FUNCTION_BLOCK FlushGritScreenCond (* Basic Function Block Type *)
  (* Standard: 61499-2 *)
  (* Version 0.0, 5/26/2024, SESA713705, Schneider Electric, Template *)
  PACKAGE SE.Nereda;
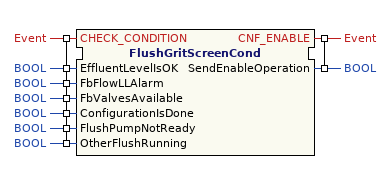
  EVENT_INPUT
    CHECK_CONDITION WITH EffluentLevelIsOK, FbFlowLLAlarm, FbValvesAvailable, ConfigurationIsDone, FlushPumpNotReady, OtherFlushRunning;
  END_EVENT
  EVENT_OUTPUT
    CNF_ENABLE WITH SendEnableOperation; (* Execution Confirmation *)
  END_EVENT
  VAR_INPUT
    EffluentLevelIsOK : BOOL;
    FbFlowLLAlarm : BOOL;
    FbValvesAvailable : BOOL;
    ConfigurationIsDone : BOOL;
    FlushPumpNotReady : BOOL;
    OtherFlushRunning : BOOL;
  END_VAR
  VAR_OUTPUT
    SendEnableOperation : BOOL;
  END_VAR
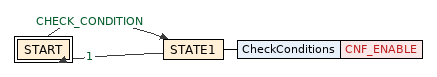
  EC_STATES
    START; (* Initial State *)
    STATE1 : CheckConditions -> CNF_ENABLE;
  END_STATES
  EC_TRANSITIONS
    START TO STATE1 := CHECK_CONDITION;
    STATE1 TO START := 1;
  END_TRANSITIONS
  ALGORITHM CheckConditions IN ST:
;
IF 	EffluentLevelIsOK = TRUE AND
	FbFlowLLAlarm = FALSE AND
	FbValvesAvailable = TRUE AND
	NOT OtherFlushRunning AND
	ConfigurationIsDone = TRUE AND
	FlushPumpNotReady = FALSE THEN

	SendEnableOperation := TRUE;
ELSE
	SendEnableOperation := FALSE;
END_IF;
  END_ALGORITHM
END_FUNCTION_BLOCK
